// One sink standing for many. A suite holds a single I_TestReporter and never
// learns how many are behind it.
//
// The composite is what makes several reporting problems disappear
// rather than get solved. The individual re-run that "records nothing and saves
// nothing" becomes a matter of NOT CALLING this object, rather than a flag
// threaded through the runner. Severity policy and the duplicated event-logger
// blocks become choices about which sinks a build attaches.
//
// It can also be SUSPENDED, which is what makes an individual re-run possible
// without a condition threaded through the runner.
//
// It implements I_TestDetailSink as well, and fans checks out only to the sinks
// that wanted them. Each reporter is queried once, when it is attached; a
// per-check query would put an interface lookup in the hottest path in the
// library.
//
// Not generic. Its capacity is a parameter rather than a generic argument because
// a project attaches the same set of sinks to every suite it owns, so per-instance
// variation would cost every declaration site an argument to buy nothing.
FUNCTION_BLOCK TestReporterFanout IMPLEMENTS I_TestReporter, I_TestDetailSink
VAR
	_Reporters : ARRAY[0..TestHarnessParameter.ReporterCapacity - 1] OF I_TestReporter;
	// Parallel to _Reporters: element i is the detail face of reporter i, or null
	// where that reporter did not want checks. Resolved once, at Add.
	_DetailSinks : ARRAY[0..TestHarnessParameter.ReporterCapacity - 1] OF I_TestDetailSink;
	_Count : UDINT;

	// While TRUE, notifications are dropped and nothing reaches a sink.
	//
	// This is how an individual re-run records nothing and saves nothing: the suite
	// silences every sink at once, rather than a condition threaded through the
	// runner and the journal and remembered in three places.
	//
	// CyclicLogic is NOT suppressed. A file write already in flight must still
	// finish, or IsIdle never goes TRUE and CI waits forever.
	_IsSuspended : BOOL;
END_VAR

(*
	No cyclic body of its own. CyclicLogic is the cyclic entry point and is called
	by the suite, which is itself driven.
*)

// Attach a sink. Order of attachment is order of notification.
//
// Not named Add: ADD is a standard function and TwinCAT is case-insensitive.
//
// Every reporter attached receives everything; there is no filtering here, because
// a sink that wants less can decide that for itself.
//
// A reporter is queried ONCE for I_TestDetailSink and the answer is stored. A
// per-check __QUERYINTERFACE would put an interface lookup inside the hottest path
// in the library - a forty-check test would pay for forty of them.
//
// Returns FALSE when the list is full or the reporter is null, and raises a
// framework error through the sinks ALREADY attached. That is not circular: the
// ones already there are exactly the ones that can still report it.
METHOD Attach : BOOL
VAR_INPUT
	Reporter : I_TestReporter;
END_VAR

VAR
	Index : DINT;
END_VAR
Attach := FALSE;

IF Reporter = 0 THEN
	THIS^.FrameworkError('TestReporterFanout', 'a null reporter was offered');
	RETURN;
END_IF

IF _Count >= TestHarnessParameter.ReporterCapacity THEN
	THIS^.FrameworkError('TestReporterFanout',
		'reporter list is full - raise TestHarnessParameter.ReporterCapacity');
	RETURN;
END_IF

Index := TO_DINT(_Count);

_Reporters[Index] := Reporter;

// Optional, exactly as the test hooks are. A sink that only wants verdicts does
// not implement it and is never called for checks.
IF NOT __QUERYINTERFACE(Reporter, _DetailSinks[Index]) THEN
	_DetailSinks[Index] := 0;
END_IF

_Count := _Count + 1;
Attach := TRUE;
END_METHOD

METHOD CheckFailed
VAR_INPUT
	StepLabel  : T_MaxString;
	Kind	   : E_FailureKind;
	Expected   : T_MaxString;
	Actual	   : T_MaxString;
	Diagnostic : T_MaxString;
	Message	   : T_MaxString;
END_VAR

VAR
	i : DINT;
END_VAR
IF _IsSuspended THEN
	RETURN;
END_IF

FOR i := 0 TO TO_DINT(_Count) - 1 DO
	IF _DetailSinks[i] <> 0 THEN
		_DetailSinks[i].CheckFailed(
			StepLabel  := StepLabel,
			Kind	   := Kind,
			Expected   := Expected,
			Actual	   := Actual,
			Diagnostic := Diagnostic,
			Message	   := Message);
	END_IF
END_FOR
END_METHOD

METHOD CheckPassed
VAR_INPUT
	StepLabel : T_MaxString;
	Detail	  : T_MaxString;
END_VAR

VAR
	i : DINT;
END_VAR
IF _IsSuspended THEN
	RETURN;
END_IF

FOR i := 0 TO TO_DINT(_Count) - 1 DO
	IF _DetailSinks[i] <> 0 THEN
		_DetailSinks[i].CheckPassed(StepLabel := StepLabel, Detail := Detail);
	END_IF
END_FOR
END_METHOD

// Sinks attached. Assert it in CI: a reporter that silently stops being attached
// takes its output with it, and a result file that never appears reads as a broken
// build rather than as a missing sink.
PROPERTY Count : UDINT
GET
Count := _Count;
END_GET
END_PROPERTY

// Advance every sink, every scan, unconditionally.
//
// This is what lets a reporter be slow without blocking a test. Anything that
// takes time - a file write, an ADS call - is STARTED in one of the notification
// methods and ADVANCED here.
METHOD CyclicLogic
VAR
	i : DINT;
END_VAR
FOR i := 0 TO TO_DINT(_Count) - 1 DO
	_Reporters[i].CyclicLogic();
END_FOR
END_METHOD

// Never silent, and never reported as a test failure.
//
// Reaching here with nothing attached IS silent, and there is nothing this object
// can do about it. That is what ReporterCount exists for: assert it in CI.
METHOD FrameworkError
VAR_INPUT
	Source	: T_MaxString;
	Message : T_MaxString;
END_VAR

VAR
	i : DINT;
END_VAR
IF _IsSuspended THEN
	RETURN;
END_IF

FOR i := 0 TO TO_DINT(_Count) - 1 DO
	_Reporters[i].FrameworkError(Source := Source, Message := Message);
END_FOR
END_METHOD

// FALSE while ANY attached sink still has work in flight.
//
// CI must wait for this as well as IsComplete. A run finishing and its result
// document reaching disk are different events, and copying between them yields a
// truncated artifact - which reads as a broken pipeline rather than a finished
// run.
//
// TRUE with nothing attached: no sink, no pending work.
PROPERTY IsIdle : BOOL
GET
VAR
	i : DINT;
END_VAR
IsIdle := TRUE;

FOR i := 0 TO TO_DINT(_Count) - 1 DO
	IF NOT _Reporters[i].IsIdle THEN
		IsIdle := FALSE;
		RETURN;
	END_IF
END_FOR
END_GET
END_PROPERTY

// Notify sinks again. Nothing that happened while suspended is replayed - it was
// deliberately not recorded.
METHOD Resume
_IsSuspended := FALSE;
END_METHOD

METHOD RunFinished
VAR_INPUT
	Status	   : I_TestRunStatus;
	TargetInfo : T_MaxString;
END_VAR

VAR
	i : DINT;
END_VAR
IF _IsSuspended THEN
	RETURN;
END_IF

FOR i := 0 TO TO_DINT(_Count) - 1 DO
	_Reporters[i].RunFinished(Status := Status, TargetInfo := TargetInfo);
END_FOR
END_METHOD

METHOD RunStarted
VAR_INPUT
	Label	   : T_MaxString;
	TargetInfo : T_MaxString;
END_VAR

VAR
	i : DINT;
END_VAR
IF _IsSuspended THEN
	RETURN;
END_IF

FOR i := 0 TO TO_DINT(_Count) - 1 DO
	_Reporters[i].RunStarted(Label := Label, TargetInfo := TargetInfo);
END_FOR
END_METHOD

METHOD SuiteFinished
VAR_INPUT
	Status : I_TestRunStatus;
END_VAR

VAR
	i : DINT;
END_VAR
IF _IsSuspended THEN
	RETURN;
END_IF

FOR i := 0 TO TO_DINT(_Count) - 1 DO
	_Reporters[i].SuiteFinished(Status);
END_FOR
END_METHOD

// Stop notifying sinks. Used for an individual re-run, which must not pollute the
// CI artifact with duplicate entries.
//
// Work already in flight is unaffected - CyclicLogic keeps running - so a document
// being written when this is called still lands.
METHOD Suspend
_IsSuspended := TRUE;
END_METHOD

METHOD TestFinished
VAR_INPUT
	SuiteLabel	  : T_MaxString;
	TestLabel	  : T_MaxString;
	Location	  : T_MaxString;
	Status		  : E_TestStatus;
	Kind		  : E_FailureKind;
	Summary		  : T_MaxString;
	ElapsedTime	  : LREAL;
	ElapsedCycles : UDINT;
	Assertions	  : UDINT;
END_VAR

VAR
	i : DINT;
END_VAR
IF _IsSuspended THEN
	RETURN;
END_IF

FOR i := 0 TO TO_DINT(_Count) - 1 DO
	_Reporters[i].TestFinished(
		SuiteLabel	  := SuiteLabel,
		TestLabel	  := TestLabel,
		Location	  := Location,
		Status		  := Status,
		Kind		  := Kind,
		Summary		  := Summary,
		ElapsedTime	  := ElapsedTime,
		ElapsedCycles := ElapsedCycles,
		Assertions	  := Assertions);
END_FOR
END_METHOD

// Only the sinks that asked for checks. A reporter that does not implement
// I_TestDetailSink is skipped without a query and without an empty method body.
METHOD TestStarted
VAR_INPUT
	SuiteLabel : T_MaxString;
	TestLabel  : T_MaxString;
	Location   : T_MaxString;
END_VAR

VAR
	i : DINT;
END_VAR
IF _IsSuspended THEN
	RETURN;
END_IF

FOR i := 0 TO TO_DINT(_Count) - 1 DO
	IF _DetailSinks[i] <> 0 THEN
		_DetailSinks[i].TestStarted(
			SuiteLabel := SuiteLabel,
			TestLabel  := TestLabel,
			Location   := Location);
	END_IF
END_FOR
END_METHOD

END_FUNCTION_BLOCK

(* stored: Version 1.1.0.1, ProductVersion 3.1.4026.18
   POU TestReporterFanout: Id {30abd70b-6653-40e9-af76-d22c0889291a}, SpecialFunc None
   Folder I_Cyclic: Id {0f6988cb-f17e-4951-b581-19b561a440fc}
   Folder I_TestDetailSink: Id {ab42cded-5788-477b-bcf8-0da4e1c521a4}
   Folder I_TestReporter: Id {5044e5ed-ab27-4794-a370-5c71587806e4}
   Method Attach: Id {b4759758-ca0f-4d90-a4e8-605ebe108d8f}
   Method CheckFailed: Id {486712c9-5282-4fe9-93a6-f73c3896a540}
   Method CheckPassed: Id {9c4e2785-3045-4687-a782-36da70ee5ef7}
   Property Count: Id {5dad202d-a9f6-4b20-9853-cafdeeac4cb2}
   Get Get: Id {f0df57ba-ead5-4c72-83c7-79a383abd884}
   Method CyclicLogic: Id {73def0a4-f0e7-4219-ad74-2768a6af2b00}
   Method FrameworkError: Id {3d5a9b01-6f7e-447f-8dd1-2cd1080080ac}
   Property IsIdle: Id {019cc85e-9e39-4f15-98db-4010e86769f3}
   Get Get: Id {f2dcf839-ea43-4546-b68f-f5b1539979c7}
   Method Resume: Id {cb881c75-5c35-4306-9969-7f2b54c8d920}
   Method RunFinished: Id {d445a976-1d73-4d95-a2a1-4bf7d7a18389}
   Method RunStarted: Id {a05a752c-c027-46c5-ab84-9d40fad541b8}
   Method SuiteFinished: Id {ec2bc5be-0df1-47a7-b8d1-031dba4bb8b1}
   Method Suspend: Id {59f8506e-4c82-4dfd-a387-7ea12c318327}
   Method TestFinished: Id {a43a6462-1cf7-4709-9ec5-69542ac23a66}
   Method TestStarted: Id {7122bfc6-401f-48e1-bc9c-c445aa5e0b97} *)
